(* CODESYS project Lark_Sheeta_VFDComm.project
   Title: Lark_Sheeta_VFDComm
   Version: 0.0.0.0

Project tree, tasks and I/O mapping:
  MyController : TM218LDAE24DRHN, Schneider Electric, order no. TM218LDAE24DRHN, version 4.0.1.26
    application Application
      task MAST (cyclic, interval 20 ms, priority 15, watchdog 100 ms x 1) calls MyPOU
      function HiddenPOU [ST]
      global variables GVL
      program MyPOU [FBD]
    Embedded Functions
      IO : IO, Schneider Electric, version 4.0.1.26
          input  iwIO_IW0 : WORD  // IW0
          output qwIO_QW0 : WORD  // QW0
      HSC : HSC, Schneider Electric, version 4.0.1.26
    Serial Line 1
      SoMachine_Network_Manager : SoMachine-Network Manager, Schneider Electric, version 4.0.0.2
    Serial Line 2
      Modbus_Manager : Modbus Manager, Schneider Electric, version 4.0.0.2
    Ethernet
        settings: IPAddress = [192, 168, 3, 20]; SubnetMask = [255, 255, 255, 0]; GatewayAddress = [192, 168, 3, 1]; WebServer = FALSE; FTP Server = FALSE; SoMachine Protocol = TRUE; Modbus Server = TRUE; NetManage Protocol = FALSE; SNMP protocol = FALSE; Enable Routing = FALSE
*)

// MyController/Application/GVL
VAR_GLOBAL
	v1Cmd AT %MW0: INT;
	v1Ref AT %MW1: INT;
	v1Stat AT %MW20: INT;
	v1RPM AT %MW21: INT;
	
	v2Cmd AT %MW2: INT;
	v2Ref AT %MW3: INT;
	v2Stat AT %MW22: INT;
	v2RPM AT %MW23: INT;
	
	v3Cmd AT %MW4: INT;
	v3Ref AT %MW5: INT;
	v3Stat AT %MW24: INT;
	v3RPM AT %MW25: INT;
	
	v4Cmd AT %MW6: INT;
	v4Ref AT %MW7: INT;
	v4Stat AT %MW26: INT;
	v4RPM AT %MW27: INT;
	
	v5Cmd AT %MW8: INT;
	v5Ref AT %MW9: INT;
	v5Stat AT %MW28: INT;
	v5RPM AT %MW29: INT;
	
	v6Cmd AT %MW10: INT;
	v6Ref AT %MW11: INT;
	v6Stat AT %MW30: INT;
	v6RPM AT %MW31 : INT;
END_VAR

// MyController/Application/MyPOU
PROGRAM MyPOU
VAR
	ADDM_0: ADDM;
	vfd1: ADDRESS;
	BLINK_0: BLINK;
	WRITE_READ_VAR_0: WRITE_READ_VAR;
	write1: ARRAY[0..1] OF WORD;
	read1: ARRAY[0..1] OF WORD;
	vfd1Done: BOOL;
	vfd1Err: BOOL;
	ADDM_1: ADDM;
	WRITE_READ_VAR_1: WRITE_READ_VAR;
	vfd2: ADDRESS;
	vfd2Done: BOOL;
	vfd2Err: BOOL;
	write2: ARRAY[0..1] OF WORD;
	read2: ARRAY[0..1] OF WORD;
	
	ADDM_2: ADDM;
	WRITE_READ_VAR_2: WRITE_READ_VAR;
	vfd3: ADDRESS;
	vfd3Done: BOOL;
	vfd3Err: BOOL;
	write3: ARRAY[0..1] OF WORD;
	read3: ARRAY[0..1] OF WORD;
	
	ADDM_3: ADDM;
	WRITE_READ_VAR_3: WRITE_READ_VAR;
	vfd4: ADDRESS;
	vfd4Done: BOOL;
	vfd4Err: BOOL;
	write4: ARRAY[0..1] OF WORD;
	read4: ARRAY[0..1] OF WORD;
	
	ADDM_4: ADDM;
	WRITE_READ_VAR_4: WRITE_READ_VAR;
	vfd5: ADDRESS;
	vfd5Done: BOOL;
	vfd5Err: BOOL;
	write5: ARRAY[0..1] OF WORD;
	read5: ARRAY[0..1] OF WORD;
	
	ADDM_5: ADDM;
	WRITE_READ_VAR_5: WRITE_READ_VAR;
	vfd6: ADDRESS;
	vfd6Done: BOOL;
	vfd6Err: BOOL;
	write6: ARRAY[0..1] OF WORD;
	read6: ARRAY[0..1] OF WORD;
	READ_VAR_0: READ_VAR;
	startCmd: WORD;
END_VAR

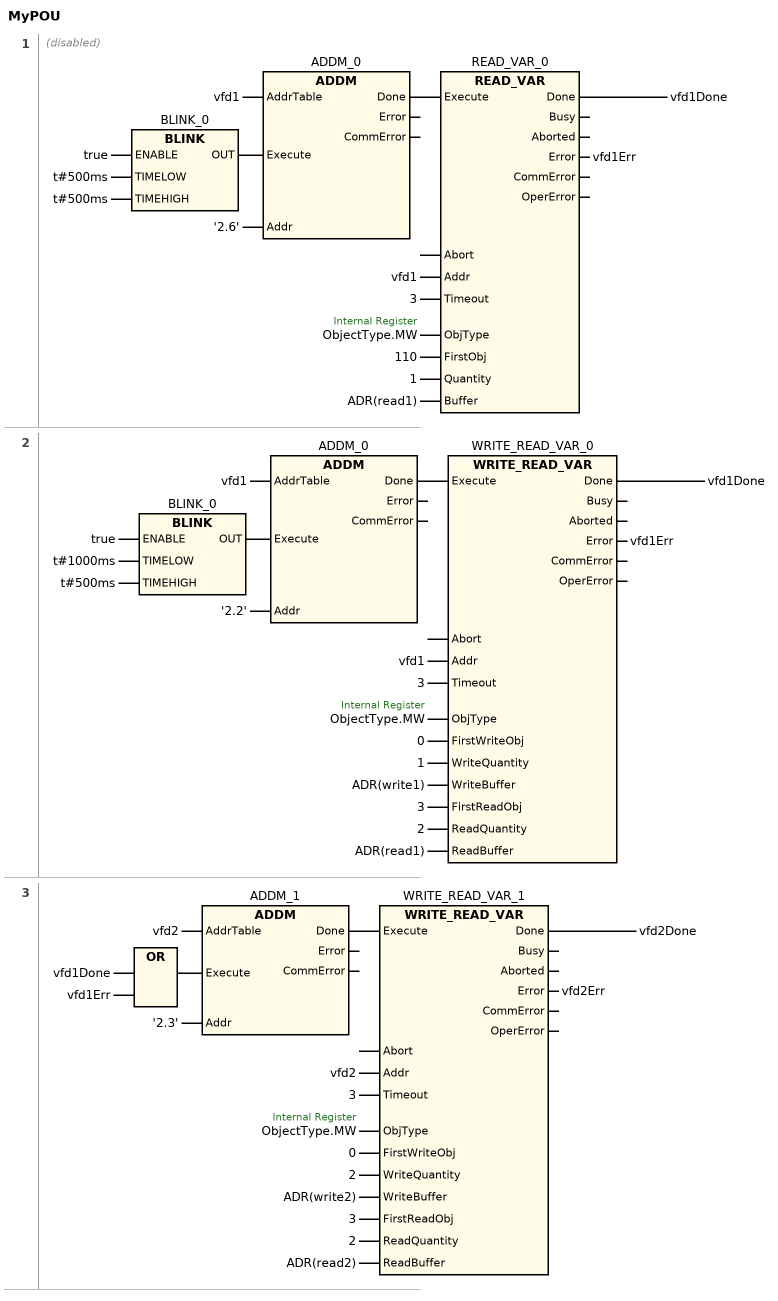
// NETWORK 1 (disabled)
//   ObjectType.MW: Internal Register
// BLINK_0(ENABLE := true, TIMELOW := t#500ms, TIMEHIGH := t#500ms); // BLINK
// ADDM_0(AddrTable := vfd1, Execute := BLINK_0.OUT, Addr := '2.6'); // ADDM
// READ_VAR_0(
//     Execute := ADDM_0.Done,
//     Addr := vfd1,
//     Timeout := 3,
//     ObjType := ObjectType.MW,
//     FirstObj := 110,
//     Quantity := 1,
//     Buffer := ADR(read1),
//     Error => vfd1Err); // READ_VAR
// vfd1Done := READ_VAR_0.Done;

// NETWORK 2
//   ObjectType.MW: Internal Register
BLINK_0(ENABLE := true, TIMELOW := t#1000ms, TIMEHIGH := t#500ms); // BLINK
ADDM_0(AddrTable := vfd1, Execute := BLINK_0.OUT, Addr := '2.2'); // ADDM
WRITE_READ_VAR_0(
    Execute := ADDM_0.Done,
    Addr := vfd1,
    Timeout := 3,
    ObjType := ObjectType.MW,
    FirstWriteObj := 0,
    WriteQuantity := 1,
    WriteBuffer := ADR(write1),
    FirstReadObj := 3,
    ReadQuantity := 2,
    ReadBuffer := ADR(read1),
    Error => vfd1Err); // WRITE_READ_VAR
vfd1Done := WRITE_READ_VAR_0.Done;

// NETWORK 3
//   ObjectType.MW: Internal Register
ADDM_1(AddrTable := vfd2, Execute := vfd1Done OR vfd1Err, Addr := '2.3'); // ADDM
WRITE_READ_VAR_1(
    Execute := ADDM_1.Done,
    Addr := vfd2,
    Timeout := 3,
    ObjType := ObjectType.MW,
    FirstWriteObj := 0,
    WriteQuantity := 2,
    WriteBuffer := ADR(write2),
    FirstReadObj := 3,
    ReadQuantity := 2,
    ReadBuffer := ADR(read2),
    Error => vfd2Err); // WRITE_READ_VAR
vfd2Done := WRITE_READ_VAR_1.Done;

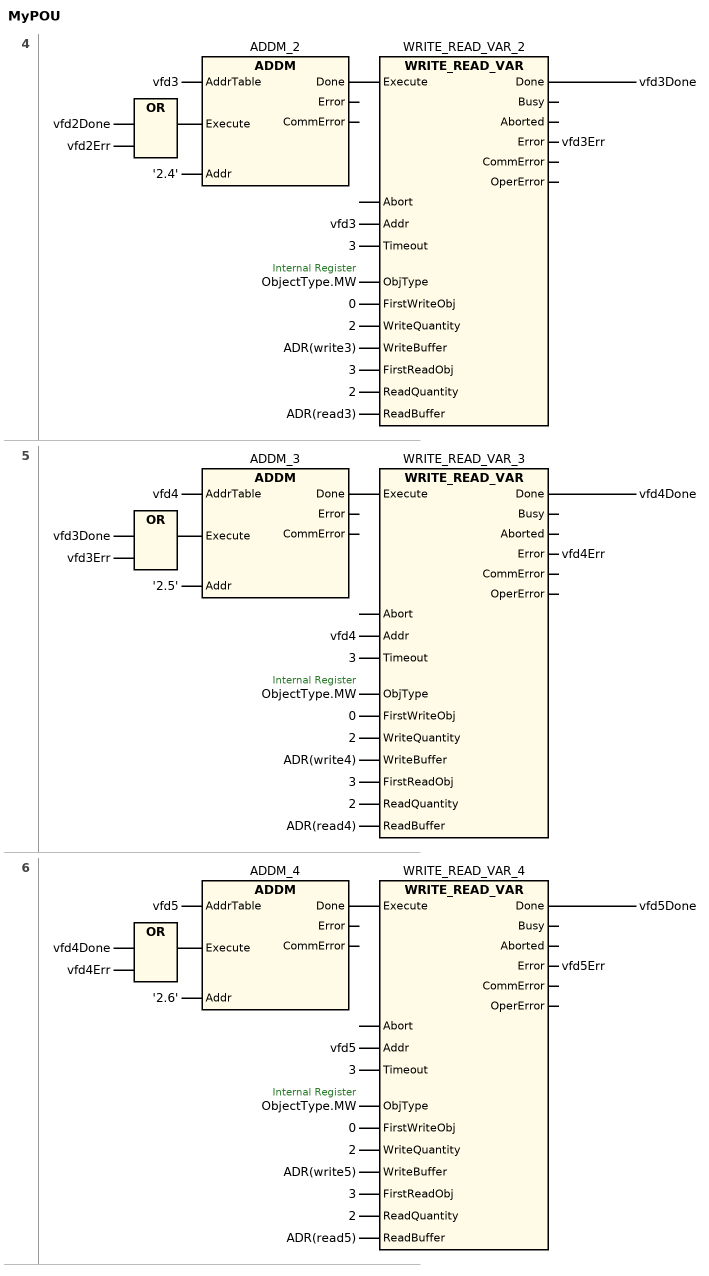
// NETWORK 4
//   ObjectType.MW: Internal Register
ADDM_2(AddrTable := vfd3, Execute := vfd2Done OR vfd2Err, Addr := '2.4'); // ADDM
WRITE_READ_VAR_2(
    Execute := ADDM_2.Done,
    Addr := vfd3,
    Timeout := 3,
    ObjType := ObjectType.MW,
    FirstWriteObj := 0,
    WriteQuantity := 2,
    WriteBuffer := ADR(write3),
    FirstReadObj := 3,
    ReadQuantity := 2,
    ReadBuffer := ADR(read3),
    Error => vfd3Err); // WRITE_READ_VAR
vfd3Done := WRITE_READ_VAR_2.Done;

// NETWORK 5
//   ObjectType.MW: Internal Register
ADDM_3(AddrTable := vfd4, Execute := vfd3Done OR vfd3Err, Addr := '2.5'); // ADDM
WRITE_READ_VAR_3(
    Execute := ADDM_3.Done,
    Addr := vfd4,
    Timeout := 3,
    ObjType := ObjectType.MW,
    FirstWriteObj := 0,
    WriteQuantity := 2,
    WriteBuffer := ADR(write4),
    FirstReadObj := 3,
    ReadQuantity := 2,
    ReadBuffer := ADR(read4),
    Error => vfd4Err); // WRITE_READ_VAR
vfd4Done := WRITE_READ_VAR_3.Done;

// NETWORK 6
//   ObjectType.MW: Internal Register
ADDM_4(AddrTable := vfd5, Execute := vfd4Done OR vfd4Err, Addr := '2.6'); // ADDM
WRITE_READ_VAR_4(
    Execute := ADDM_4.Done,
    Addr := vfd5,
    Timeout := 3,
    ObjType := ObjectType.MW,
    FirstWriteObj := 0,
    WriteQuantity := 2,
    WriteBuffer := ADR(write5),
    FirstReadObj := 3,
    ReadQuantity := 2,
    ReadBuffer := ADR(read5),
    Error => vfd5Err); // WRITE_READ_VAR
vfd5Done := WRITE_READ_VAR_4.Done;

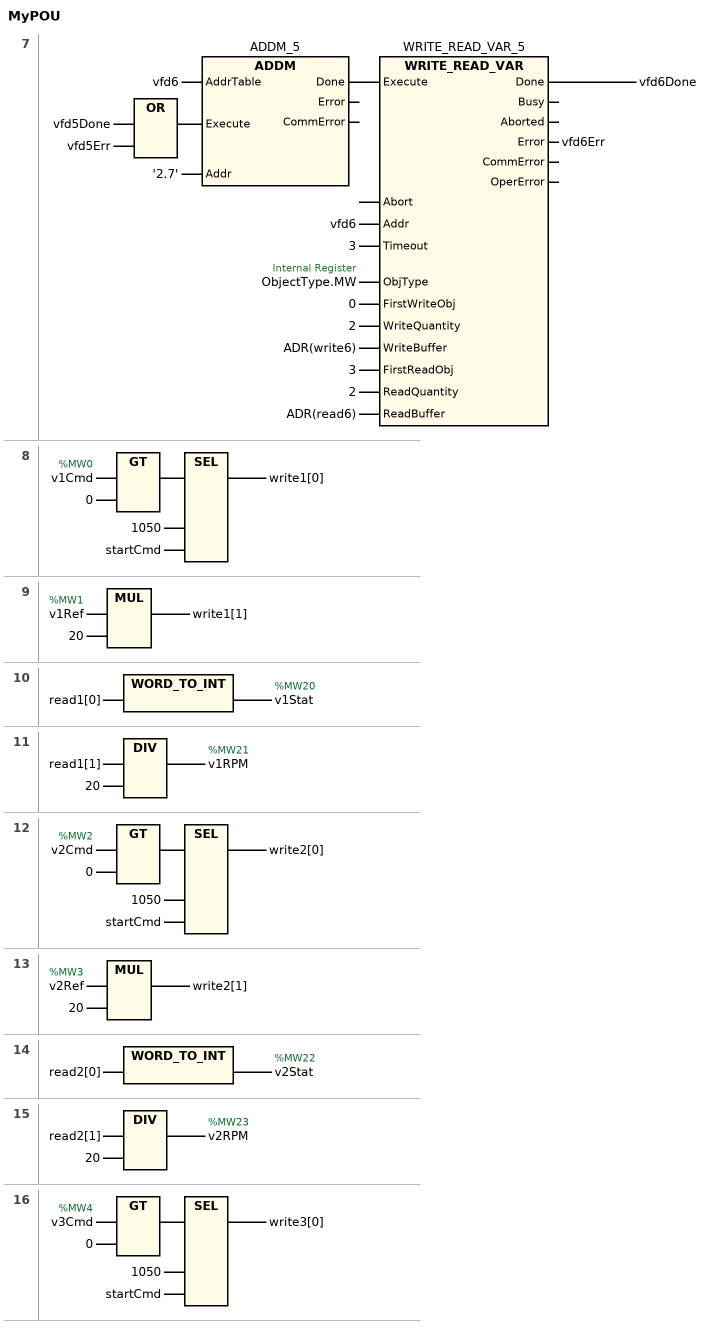
// NETWORK 7
//   ObjectType.MW: Internal Register
ADDM_5(AddrTable := vfd6, Execute := vfd5Done OR vfd5Err, Addr := '2.7'); // ADDM
WRITE_READ_VAR_5(
    Execute := ADDM_5.Done,
    Addr := vfd6,
    Timeout := 3,
    ObjType := ObjectType.MW,
    FirstWriteObj := 0,
    WriteQuantity := 2,
    WriteBuffer := ADR(write6),
    FirstReadObj := 3,
    ReadQuantity := 2,
    ReadBuffer := ADR(read6),
    Error => vfd6Err); // WRITE_READ_VAR
vfd6Done := WRITE_READ_VAR_5.Done;

// NETWORK 8
//   v1Cmd: AT %MW0
write1[0] := SEL(v1Cmd > 0, 1050, startCmd);

// NETWORK 9
//   v1Ref: AT %MW1
write1[1] := v1Ref * 20;

// NETWORK 10
//   v1Stat: AT %MW20
v1Stat := WORD_TO_INT(read1[0]);

// NETWORK 11
//   v1RPM: AT %MW21
v1RPM := read1[1] / 20;

// NETWORK 12
//   v2Cmd: AT %MW2
write2[0] := SEL(v2Cmd > 0, 1050, startCmd);

// NETWORK 13
//   v2Ref: AT %MW3
write2[1] := v2Ref * 20;

// NETWORK 14
//   v2Stat: AT %MW22
v2Stat := WORD_TO_INT(read2[0]);

// NETWORK 15
//   v2RPM: AT %MW23
v2RPM := read2[1] / 20;

// NETWORK 16
//   v3Cmd: AT %MW4
write3[0] := SEL(v3Cmd > 0, 1050, startCmd);

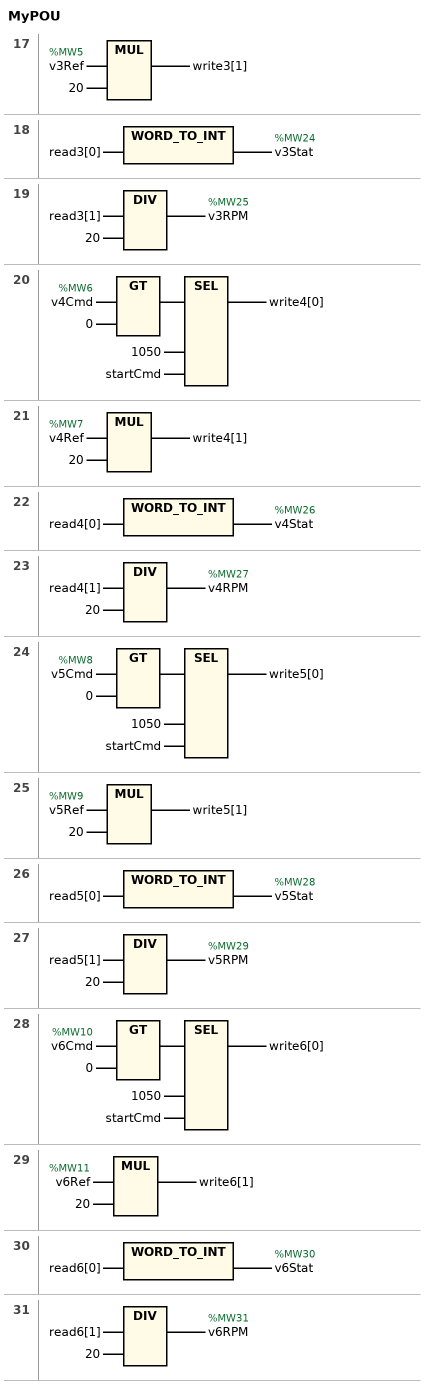
// NETWORK 17
//   v3Ref: AT %MW5
write3[1] := v3Ref * 20;

// NETWORK 18
//   v3Stat: AT %MW24
v3Stat := WORD_TO_INT(read3[0]);

// NETWORK 19
//   v3RPM: AT %MW25
v3RPM := read3[1] / 20;

// NETWORK 20
//   v4Cmd: AT %MW6
write4[0] := SEL(v4Cmd > 0, 1050, startCmd);

// NETWORK 21
//   v4Ref: AT %MW7
write4[1] := v4Ref * 20;

// NETWORK 22
//   v4Stat: AT %MW26
v4Stat := WORD_TO_INT(read4[0]);

// NETWORK 23
//   v4RPM: AT %MW27
v4RPM := read4[1] / 20;

// NETWORK 24
//   v5Cmd: AT %MW8
write5[0] := SEL(v5Cmd > 0, 1050, startCmd);

// NETWORK 25
//   v5Ref: AT %MW9
write5[1] := v5Ref * 20;

// NETWORK 26
//   v5Stat: AT %MW28
v5Stat := WORD_TO_INT(read5[0]);

// NETWORK 27
//   v5RPM: AT %MW29
v5RPM := read5[1] / 20;

// NETWORK 28
//   v6Cmd: AT %MW10
write6[0] := SEL(v6Cmd > 0, 1050, startCmd);

// NETWORK 29
//   v6Ref: AT %MW11
write6[1] := v6Ref * 20;

// NETWORK 30
//   v6Stat: AT %MW30
v6Stat := WORD_TO_INT(read6[0]);

// NETWORK 31
//   v6RPM: AT %MW31
v6RPM := read6[1] / 20;

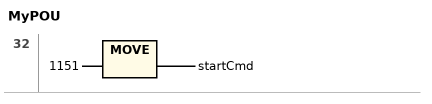
// NETWORK 32
startCmd := 1151;

END_PROGRAM

// MyController/Application/HiddenPOU
FUNCTION HiddenPOU : BOOL

VAR_INPUT
	pHiddenFunc: POINTER TO WORD;
END_VAR
VAR
	pRead: POINTER TO BYTE;
	pWrite: POINTER TO BYTE;
END_VAR

pRead := pHiddenFunc + 400;
pWrite := pHiddenFunc + 4400;
HiddenPOU := TRUE;

END_FUNCTION
